PROGRAM AxisCaliHomePos
VAR
	writeParam		:MC_WriteParameter;
	bWriteParam_DO	:BOOL;
	
END_VAR


writeParam(
	Axis:= axis_RightArm_Wrist, 
	Execute:= bWriteParam_DO, 
	ParameterNumber:= AxisEncoderOffset, 
	Value:= -2, 
	Done=> , 
	Busy=> , 
	Error=> , 
	ErrorID=> );

END_PROGRAM

(* stored: Version 1.1.0.1, ProductVersion 3.1.4024.14
   POU AxisCaliHomePos: Id {eb4c649f-b337-425e-8072-20a3a253b07a}, SpecialFunc None *)
